Staubli VAL3: onEnterEvent.pgx

program onEnterEvent(bool& x_bSave[])
  local bool l_bOk
begin
  //
  // NB sEvent is the selected
  // element in the LIST
  //
  call use:stringToArray(sTrajName+","+toString("",nIndex),sMessage)
  // update all

  call loadPage("Disk://trajectory/page_editTraj",sMessage)
  // ELEBORATE THE GIVE BACK
  //
  if sMessage[0]=="saved"
    sItems[0]="saved"
    x_bSave=false
  endIf
  l_bOk=true
  toNum(sMessage[1],nSelect,l_bOk)
  // reset the show status
  bShowStatus=false
end
